FUNCTION_BLOCK counter
VAR
    counter : DINT; 
END_VAR

counter := counter + 1;

METHOD FB_init : BOOL
VAR_INPUT
	bInitRetains : BOOL; // if TRUE, the retain variables are initialized (warm start / cold start)
	bInCopyCode : BOOL;  // if TRUE, the instance afterwards gets moved into the copy code (online change)
    start : DINT;
END_VAR
counter := start;
END_METHOD

{attribute 'monitoring' := 'call'}
{attribute 'TcRpcEnable'}
PROPERTY Value : DINT
GET
Value := THIS^.counter;
END_GET
SET
THIS^.counter := Value;
END_SET
END_PROPERTY

END_FUNCTION_BLOCK

(* stored: Version 1.1.0.1, ProductVersion 3.1.4024.12
   POU counter: Id {4794190c-2183-498f-9e08-a352c9417c87}, SpecialFunc None
   Method FB_init: Id {6136ff50-caf9-4e9d-bf15-6f8696783c81}
   Property Value: Id {fe35c301-dd46-43cd-90b4-572e272cf8ae}
   Get Get: Id {edc70f8b-9e7e-4de5-8974-10b8a534f7fd}
   Set Set: Id {61f3337d-7662-4a91-ab34-1f98c1964bda} *)
